FUNCTION_BLOCK FB_Axis_HomeToSensor EXTENDS FB_AxisBase
VAR_INPUT
END_VAR
VAR_OUTPUT
END_VAR
VAR
	//I/O definitions
	fbHomeSensor		: FB_Sensor;
	
	//Internal Property Variables
	fHomePositionSetpoint		: LREAL := 0;
	bHomeSensorStatus			: BOOL;
END_VAR

METHOD Home : BOOL
VAR_INPUT
END_VAR
SUPER^.Home();

IF NOT bActive THEN
	fbAxisHome.Execute := TRUE;
END_IF
END_METHOD

PROPERTY HomePositionSetpoint : LREAL
GET
HomePositionSetpoint := fHomePositionSetpoint;
END_GET
SET
fHomePositionSetpoint := HomePositionSetpoint;
END_SET
END_PROPERTY

PROPERTY HomeSensorStatus : BOOL
GET
HomeSensorStatus := bHomeSensorStatus;
END_GET
END_PROPERTY

METHOD Monitoring : BOOL
SUPER^.Monitoring();

bHomeSensorStatus := fbHomeSensor.Active;
END_METHOD

METHOD MotionControl : BOOL
VAR_INPUT
END_VAR
SUPER^.MotionControl();

//Performs a simple home-to sensor sequence when commanded by a "Home" Method call
fbAxisHome(
	Axis:= SelectedAxis,
	Position:= fHomePositionSetpoint, 
	HomingMode:= MC_HomingMode.MC_DefaultHoming, 
	BufferMode:= MC_BufferMode.MC_Aborting,
	bCalibrationCam := bHomeSensorStatus);

fbAxisHome.Execute := FALSE;
END_METHOD

END_FUNCTION_BLOCK

(* stored: Version 1.1.0.1, ProductVersion 3.1.4024.9
   POU FB_Axis_HomeToSensor: Id {34bcfaf3-b9c7-4614-94fc-f206ca269743}, SpecialFunc None
   Folder 01_SUPER_Overrides: Id {b7e810e7-7286-4afa-9522-69b155784007}
   Method Home: Id {62fb52c0-a114-4189-a183-d55826f92029}
   Property HomePositionSetpoint: Id {db3ab09f-698b-4e2a-8d13-406e53711f63}
   Get Get: Id {33168fc0-5488-42e5-8ef0-3ae2f8d701dc}
   Set Set: Id {5c11391f-a161-4599-acac-f76ee097e0ad}
   Property HomeSensorStatus: Id {3207e959-91ef-4c72-8ae1-e13995231f9b}
   Get Get: Id {1e134f28-dfbd-47a4-9cdd-ac23a4ac4d54}
   Method Monitoring: Id {96c31064-1ccf-48ca-97bc-db381be31831}
   Method MotionControl: Id {0febfd92-be0d-4356-a3fd-12ac6da81bf1} *)
